// TIA Portal project "Betriebsstundenzähler_ST" (V16)

(* hardware
DEVICE "S7-1200 station_1"  S7-1200 Station
   slot 0: "Rack_0"  S7-1200 Rack  Rack  V1.0
   slot 1: "PLC_1"  CPU 1212C DC/DC/DC  6ES7 212-1AE40-0XB0  V4.4
*)

// ===== PLC "PLC_1"  CPU 1212C DC/DC/DC =====

VAR_GLOBAL   // PLC tag table "Default tag table"
   "Einschalttaste_Eingang" AT %I0.0 : Bool;
   "Resettaste_Eingang" AT %I0.1 : Bool;
   "Systemeinschalt_Bit" AT %M0.0 : Bool;
   "Reset_Bit" AT %M0.1 : Bool;
   "Sekunden_S" AT %MW4 : Int;
   "Sekunden_mS" AT %MD6 : DInt;
   "Minuten" AT %MW2 : Int;
   "Stunden" AT %MW10 : Int;
   "Stunden*1000" AT %MW12 : Int;
END_VAR

DATA_BLOCK "IO_DB"   // DB1
{ S7_Optimized_Access := 'TRUE' }
VERSION : 0.1
// stored: InstanceOfName IO
"IO"
BEGIN
END_DATA_BLOCK

DATA_BLOCK "Steuerlogik_DB"   // DB2
{ S7_Optimized_Access := 'TRUE' }
VERSION : 0.1
// stored: InstanceOfName Steuerlogik
"Steuerlogik"
BEGIN
END_DATA_BLOCK

// folder: System blocks/Program resources

DATA_BLOCK "Timer"   // DB3
{ S7_Optimized_Access := 'TRUE' }
AUTHOR : Simatic
FAMILY : IEC
NAME : IEC_TMR
VERSION : 1.0
// stored: InstanceOfName IEC_TIMER
"IEC_TIMER"
BEGIN
END_DATA_BLOCK

DATA_BLOCK "Minuten_Zähler"   // DB4
{ S7_Optimized_Access := 'TRUE' }
AUTHOR : Simatic
FAMILY : IEC
NAME : CNTR
VERSION : 1.0
// stored: InstanceOfName IEC_COUNTER
"IEC_COUNTER"
BEGIN
END_DATA_BLOCK

DATA_BLOCK "Stunden_Zähler"   // DB5
{ S7_Optimized_Access := 'TRUE' }
AUTHOR : Simatic
FAMILY : IEC
NAME : CNTR
VERSION : 1.0
// stored: InstanceOfName IEC_COUNTER
"IEC_COUNTER"
BEGIN
END_DATA_BLOCK

DATA_BLOCK "Stunden*1000_Zähler"   // DB6
{ S7_Optimized_Access := 'TRUE' }
AUTHOR : Simatic
FAMILY : IEC
NAME : CNTR
VERSION : 1.0
// stored: InstanceOfName IEC_COUNTER
"IEC_COUNTER"
BEGIN
END_DATA_BLOCK

// folder: (top level)

FUNCTION_BLOCK "IO"   // FB1, SCL
{ S7_Optimized_Access := 'TRUE' }
VERSION : 0.1
BEGIN
   IF "Einschalttaste_Eingang" THEN
      "Systemeinschalt_Bit" := TRUE;
   ELSE
       "Systemeinschalt_Bit" := FALSE;
   END_IF;

   IF "Resettaste_Eingang" THEN
       "Reset_Bit" := TRUE;
   ELSE
       "Reset_Bit" := FALSE;
   END_IF;
END_FUNCTION_BLOCK

FUNCTION_BLOCK "Steuerlogik"   // FB2, SCL
{ S7_Optimized_Access := 'TRUE' }
VERSION : 0.1
   VAR
      _Timer_Reset : Bool;
      _TimerDone_Bit : Bool;
      _Minuten_Reset : Bool;
      _Minuten_ZählerDone_Bit : Bool;
      _Stunden_Reset : Bool;
      Stunden_ZählerDone_Bit : Bool;
      _Stunden_1000_Reset : Bool;
      _Stunden_1000_DoneBit : Bool;
      _Reset_All : Bool;
      ONS : Bool;
   END_VAR
BEGIN
   // Steuerlogik für Sekunden
   "Timer".TONR(IN:="Systemeinschalt_Bit",
                R:=#_Timer_Reset,
                PT:=T#60S,
                Q=>#_TimerDone_Bit);
   IF "Systemeinschalt_Bit" AND "Timer".ET <> T#60S THEN
       "Sekunden_mS" := "Timer".ET;
       "Sekunden_S" := "Sekunden_mS" / 1000;
   END_IF;

   // Steuerlogik für Minuten
   "Minuten_Zähler".CTU(CU:=#_TimerDone_Bit,
                        R:=#_Minuten_Reset,
                        PV:=60,
                        Q=>#_Minuten_ZählerDone_Bit);


   IF "Minuten_Zähler".CV <> 60 THEN
       "Minuten" := "Minuten_Zähler".CV;
   END_IF;

   // Steuerlogik für Stunden
   "Stunden_Zähler".CTU(CU:=#_Minuten_ZählerDone_Bit,
                        R:=#_Stunden_Reset,
                        PV:=1000,
                        Q=>#Stunden_ZählerDone_Bit);
   IF "Stunden_Zähler".CV <>1000 THEN
       "Stunden" := "Stunden_Zähler".CV;
   END_IF;

   // Steuerlogik für Stunden*1000
   "Stunden*1000_Zähler".CTU(CU:=#Stunden_ZählerDone_Bit,
                             R:=#_Stunden_1000_Reset,
                             PV:=1000,
                             Q=>#_Stunden_1000_DoneBit);

   IF "Stunden*1000_Zähler".CV <>1000 THEN

       "Stunden*1000" := "Stunden*1000_Zähler".CV ;
   END_IF;

   // Steuerlogik für Reset
   IF "Systemeinschalt_Bit" AND "Reset_Bit" AND NOT #ONS THEN
       #_Reset_All := TRUE;
       #ONS := TRUE;
   ELSE
       #_Reset_All := FALSE;

   END_IF;
   IF NOT "Reset_Bit" THEN
       #ONS := FALSE;
   END_IF;
   IF #_TimerDone_Bit OR #_Reset_All THEN
       #_Timer_Reset := TRUE;
   ELSE
       #_Timer_Reset := FALSE;
   END_IF;
   IF #_Minuten_ZählerDone_Bit OR #_Reset_All THEN
       #_Minuten_Reset := TRUE;
   ELSE
       #_Minuten_Reset := FALSE;

   END_IF;
   IF #Stunden_ZählerDone_Bit OR #_Reset_All THEN
       #_Stunden_Reset := TRUE;
   ELSE
       #_Stunden_Reset := FALSE;

   END_IF;
   IF #_Stunden_1000_DoneBit OR #_Reset_All THEN
       #_Stunden_1000_Reset := TRUE;
   ELSE
       #_Stunden_1000_Reset := FALSE;
   END_IF;
END_FUNCTION_BLOCK

ORGANIZATION_BLOCK "Main"   // OB1, LAD, ProgramCycle
TITLE = "Main Program Sweep (Cycle)"
{ S7_Optimized_Access := 'TRUE' }
VERSION : 0.1
// PROJEKTBESCHREIBUNG:In diesem Projekt wird ein Steuerungssystem entwickelt, das die Laufzeit einer Hauptanlage erfasst. Sobald die Anlage eingeschaltet wird, beginnt der Zähler, die Betriebsdauer in Sekunden, Minuten, Hunderten und Tausenden von Stunden zu messen und in den Speicherregistern Sekunden_S, Minuten und Stunden abzulegen. Zusätzlich gibt es eine Reset-Taste, mit der der gesamte Zählerstand auf null zurückgesetzt werden kann, um eine neue Messung zu starten. Die Steuerung erfolgt über ein Einschalttaste. Solche Systeme sind essenziell, da Betriebsstunden oft als Grundlage für Wartung, Inspektion oder Garantieansprüche dienen.
// 
// TESTKRITERIEN:
// 1)Zum Starten: Führen Sie Ihr Programm in PLCSIM aus. "Sekunden_S","Minuten" und "Stunden" sollten alle auf Null stehen. Diese Werte sollten sich nicht bewegen.
// 
// 2)
// Als Nächstes erzwingen Sie den Einschalttaste_Eingang auf 1 (geschlossen). Nun sollten wir sehen, dass "Sekunden_S" akkumuliert. Es sollte immer wieder von 0 bis 59 zählen. Jedes Mal, wenn "Sekunden_S" eine Minute vollzählt, sollte "Minuten" um eins hochgehen. Irgendwann erreicht "Minuten" den Wert 59 und springt dann wieder selbst auf 0 zurück. Wenn das passiert, sollte "Stunden" um eins hochgehen. (Auch wenn wir es nicht so lange laufen lassen werden.) Nachdem "Stunden" den Wert 999 erreicht, sollte es wieder auf 0 zurückspringen und "Stunden*1000" um eins hochgehen. Und so weiter. Um zu testen, ob "Stunden" und "Stunden*1000" funktionieren, können Sie "Minuten" und "Stunden" manuell jeweils auf ihren Grenzwert setzen, um sicherzustellen, dass alles korrekt hochzählt.
// 3)
// 
// Drittens erzwingen Sie den Einschalttaste_Eingang wieder 0 (offen). Alle Ihre Akkumulatoren  sollten genau an der Stelle einfrieren, an der sie stehen.
// 
// 
// 4)Viertens erzwingen Sie den System-Run-Eingang ein letztes Mal auf 1 (geschlossen). Die Akkumulatoren sollten genau dort weiterzählen, wo sie aufgehört haben.
// 
// 
// 5)Schließlich schalten Sie Reset_Eingang EIN und dann wieder AUS. Alle Werten sollten alle auf 0 zurückgesetzt werden.
   VAR_INPUT
      Initial_Call : Bool;   // Initial call of this OB
      Remanence : Bool;   // =True, if remanent data are available
   END_VAR
BEGIN

REGION Network 1
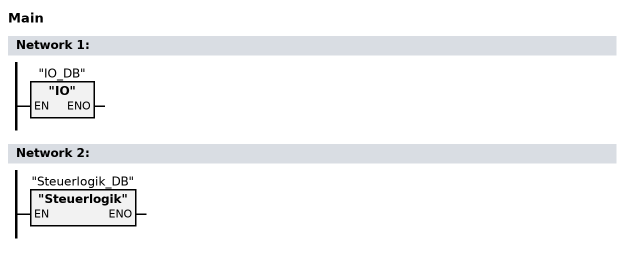
   RUNG wire#powerrail
      "IO_DB"()
   END_RUNG
   // the same network as SCL:
   "IO_DB"();   // "IO"
END_REGION

REGION Network 2
   RUNG wire#powerrail
      "Steuerlogik_DB"()
   END_RUNG
   // the same network as SCL:
   "Steuerlogik_DB"();   // "Steuerlogik"
END_REGION
END_ORGANIZATION_BLOCK